SUBAPPLICATION Uebung_123 (* Übung zu ISOBUS Name *)
  (* Standard: 61499-2; Description: Copyright (c) 2023 Meisterschulen am Ostbahnhof This program and the accompanying materials are made available under the terms of the Eclipse Public License 2.0 which is available at https://www.eclipse.org/legal/epl-2.0/ SPDX-License-Identifier: EPL-2.0 *)
  (* Version 1.0, 2023-10-23, Franz Höpfinger, Meisterschulen am Ostbahnhof, initial API and implementation and/or initial documentation *)
  PACKAGE Uebungen;
  IMPORT isobus::pgn::ISOUSERHOME_e::network;
  IMPORT isobus::pgn::ISOUSERHOME_e::thisMember;
  IMPORT isobus::pgn::ISO_CAN_NODE::NODE1;
  IMPORT Uebungen::const::Uebung_120_129::Filter::FLT_ALL_PASS;
  IMPORT Uebungen::const::Uebung_120_129::Filter::VT_ADD;
  IMPORT Uebungen::const::Uebung_120_129::Filter::VT_FLT;
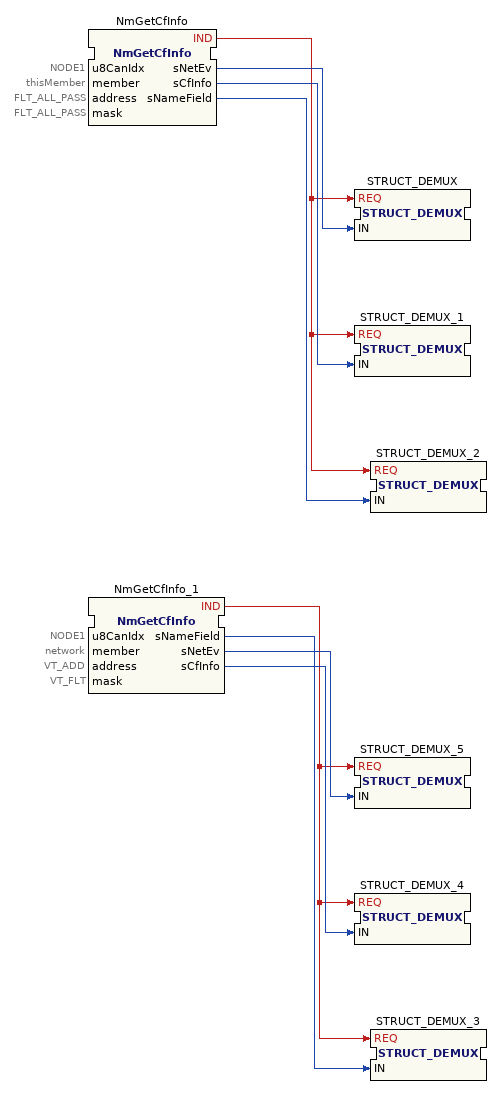
  FBS
    NmGetCfInfo : isobus::pgn::NmGetCfInfo(u8CanIdx := NODE1, member := thisMember, address := FLT_ALL_PASS, mask := FLT_ALL_PASS);
    STRUCT_DEMUX : eclipse4diac::convert::STRUCT_DEMUX; {SET_ATTRIBUTE(StructuredType, isobus::pgn::ISONETEVENT_T)}
    STRUCT_DEMUX_1 : eclipse4diac::convert::STRUCT_DEMUX; {SET_ATTRIBUTE(StructuredType, isobus::pgn::CF_INFO_T)}
    STRUCT_DEMUX_2 : eclipse4diac::convert::STRUCT_DEMUX; {SET_ATTRIBUTE(StructuredType, isobus::pgn::NAMEFIELD_T)}
    STRUCT_DEMUX_3 : eclipse4diac::convert::STRUCT_DEMUX; {SET_ATTRIBUTE(StructuredType, isobus::pgn::NAMEFIELD_T)}
    NmGetCfInfo_1 : isobus::pgn::NmGetCfInfo(u8CanIdx := NODE1, member := network, address := VT_ADD, mask := VT_FLT);
    STRUCT_DEMUX_4 : eclipse4diac::convert::STRUCT_DEMUX; {SET_ATTRIBUTE(StructuredType, isobus::pgn::CF_INFO_T)}
    STRUCT_DEMUX_5 : eclipse4diac::convert::STRUCT_DEMUX; {SET_ATTRIBUTE(StructuredType, isobus::pgn::ISONETEVENT_T)}
  END_FBS
  EVENT_CONNECTIONS
    NmGetCfInfo.IND TO STRUCT_DEMUX.REQ;
    NmGetCfInfo.IND TO STRUCT_DEMUX_1.REQ;
    NmGetCfInfo.IND TO STRUCT_DEMUX_2.REQ;
    NmGetCfInfo_1.IND TO STRUCT_DEMUX_3.REQ;
    NmGetCfInfo_1.IND TO STRUCT_DEMUX_4.REQ;
    NmGetCfInfo_1.IND TO STRUCT_DEMUX_5.REQ;
  END_CONNECTIONS
  DATA_CONNECTIONS
    NmGetCfInfo.sNetEv TO STRUCT_DEMUX.IN;
    NmGetCfInfo.sCfInfo TO STRUCT_DEMUX_1.IN;
    NmGetCfInfo.sNameField TO STRUCT_DEMUX_2.IN;
    NmGetCfInfo_1.sNameField TO STRUCT_DEMUX_3.IN;
    NmGetCfInfo_1.sNetEv TO STRUCT_DEMUX_5.IN;
    NmGetCfInfo_1.sCfInfo TO STRUCT_DEMUX_4.IN;
  END_CONNECTIONS
END_SUBAPPLICATION
